// TIA Portal V17 program export: 1 tag tables, 0 data types, 0 data blocks, 2 code blocks (in call order from the OBs), 3 instance data blocks

VAR_GLOBAL   // PLC tag table "Variablentabelle_1"
   BO AT %I20.0 : Bool;
   B1 AT %I20.1 : Bool;
   B2 AT %I20.2 : Bool;
   B3 AT %I20.3 : Bool;
   B4 AT %I20.4 : Bool;
   Rücksetztaster AT %I20.5 : Bool;
   Y1 AT %Q20.0 : Bool;
   Y2 AT %Q20.1 : Bool;
   Tag_4 AT %Q20.2 : Bool;
END_VAR

ORGANIZATION_BLOCK "Main"   // OB1, FBD, ProgramCycle
TITLE = "Main Program Sweep (Cycle)"
{ S7_Optimized_Access := 'TRUE' }
VERSION : 0.1
// stored: AutoNumber true, IsIECCheckEnabled false, SetENOAutomatically false
   VAR_INPUT
      Initial_Call : Bool;   // Initial call of this OB
      Remanence : Bool;   // =True, if remanent data are available
   END_VAR
BEGIN

REGION Network 1
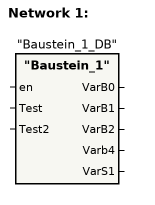
   "Baustein_1_DB"();   // "Baustein_1"
END_REGION
END_ORGANIZATION_BLOCK

FUNCTION_BLOCK "Baustein_1"   // FB1, FBD
{ S7_Optimized_Access := 'TRUE' }
VERSION : 0.1
// stored: AutoNumber true, IsIECCheckEnabled false, IsRetainMemResEnabled false, MemoryReserve 100, SetENOAutomatically false, UDAEnableTagReadback false
   VAR_OUTPUT
      VarB0 : Bool;
      VarB1 : Bool;
      VarB2 : Bool;
      Varb4 : Bool;
      VarS1 : Bool;
   END_VAR
   VAR_IN_OUT
      Test : Bool;
      Test2 : Bool;
   END_VAR
   VAR_TEMP   // added for the SCL form of the ladder/FBD networks
      _w1 : Bool;
   END_VAR
BEGIN

REGION Network 1
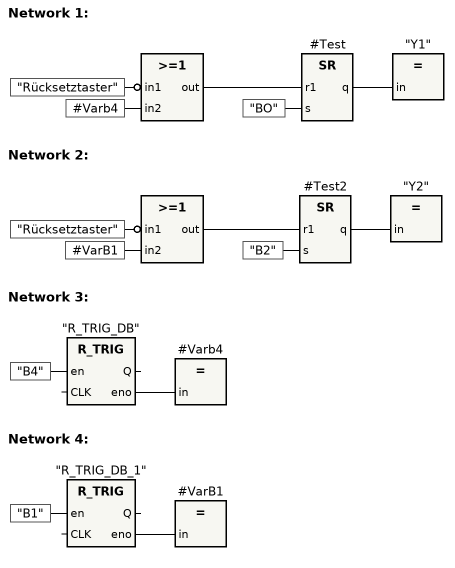
   IF "BO" THEN
       #Test := TRUE;   // SR flip-flop
   END_IF;
   IF NOT "Rücksetztaster" OR #Varb4 THEN #Test := FALSE; END_IF;
   "Y1" := #Test;
END_REGION

REGION Network 2
   IF "B2" THEN
       #Test2 := TRUE;   // SR flip-flop
   END_IF;
   IF NOT "Rücksetztaster" OR #VarB1 THEN #Test2 := FALSE; END_IF;
   "Y2" := #Test2;
END_REGION

REGION Network 3
   "R_TRIG_DB"(EN := "B4", ENO => #_w1);   // R_TRIG
   #Varb4 := #_w1;
END_REGION

REGION Network 4
   "R_TRIG_DB_1"(EN := "B1", ENO => #_w1);   // R_TRIG
   #VarB1 := #_w1;
END_REGION
END_FUNCTION_BLOCK

DATA_BLOCK "Baustein_1_DB"   // DB3
VERSION : 0.1
// stored: AutoNumber true, DBAccessibleFromOPCUA true, InstanceOfName Baustein_1, InstanceOfType FB
"Baustein_1"
BEGIN
END_DATA_BLOCK

DATA_BLOCK "R_TRIG_DB"   // DB1
// stored: AutoNumber true, DBAccessibleFromOPCUA true, InstanceOfName R_TRIG, OfSystemLibElement R_TRIG, OfSystemLibVersion 1.0
"R_TRIG"
   // VAR_INPUT
   //    CLK : Bool;
   // END_VAR
   // VAR_OUTPUT
   //    Q : Bool;
   // END_VAR
   // VAR
   //    Stat_Bit : Bool;
   // END_VAR
BEGIN
END_DATA_BLOCK

DATA_BLOCK "R_TRIG_DB_1"   // DB2
// stored: AutoNumber true, DBAccessibleFromOPCUA true, InstanceOfName R_TRIG, OfSystemLibElement R_TRIG, OfSystemLibVersion 1.0
"R_TRIG"
   // VAR_INPUT
   //    CLK : Bool;
   // END_VAR
   // VAR_OUTPUT
   //    Q : Bool;
   // END_VAR
   // VAR
   //    Stat_Bit : Bool;
   // END_VAR
BEGIN
END_DATA_BLOCK
